// Mitsubishi GX Works2 project: plc_fact_fuc_1008   PLC: Q02/Q02H

// global labels: Global1
VAR_GLOBAL
  vision AT D100 : INT;
  scan AT D102 : INT;
END_VAR

PROGRAM MAIN
VAR
  CY_1 : pusher;
  CY_2 : pusher;
  CY_3 : pusher;
END_VAR
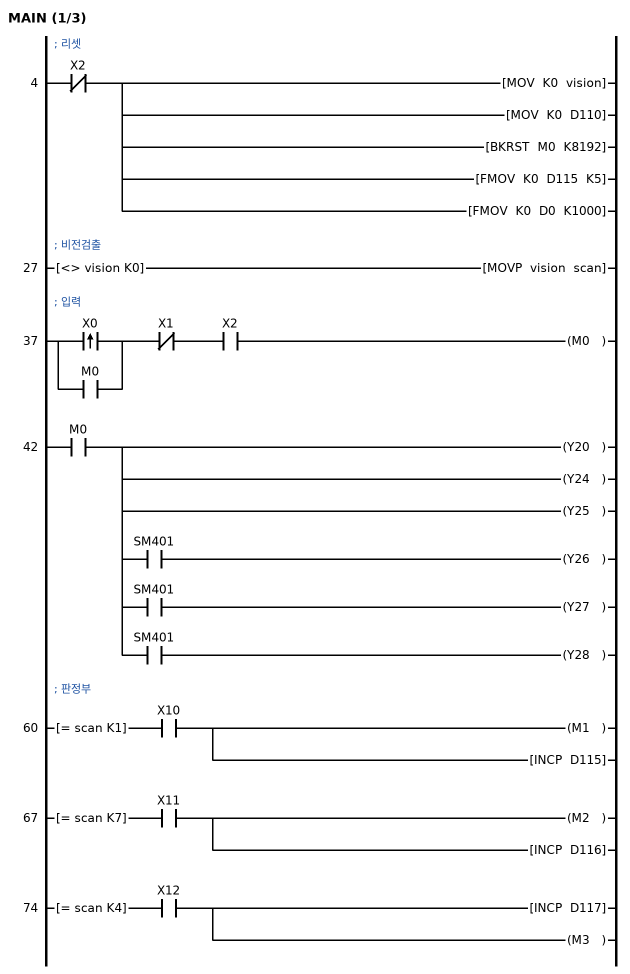
; 리셋
4     LDI     X2
      MOV     K0 vision
      MOV     K0 D110
      BKRST   M0 K8192
      FMOV    K0 D115 K5
      FMOV    K0 D0 K1000
; 비전검출
27    LD<>    vision K0
      MOVP    vision scan
; 입력
37    LDP     X0
      OR      M0
      ANI     X1
      AND     X2
      OUT     M0
42    LD      M0
      OUT     Y20
      OUT     Y24
      OUT     Y25
      MPS
      AND     SM401
      OUT     Y26
      MRD
      AND     SM401
      OUT     Y27
      MPP
      AND     SM401
      OUT     Y28
; 판정부
60    LD=     scan K1
      AND     X10
      OUT     M1
      INCP    D115
67    LD=     scan K7
      AND     X11
      OUT     M2
      INCP    D116
74    LD=     scan K4
      AND     X12
      INCP    D117
      OUT     M3
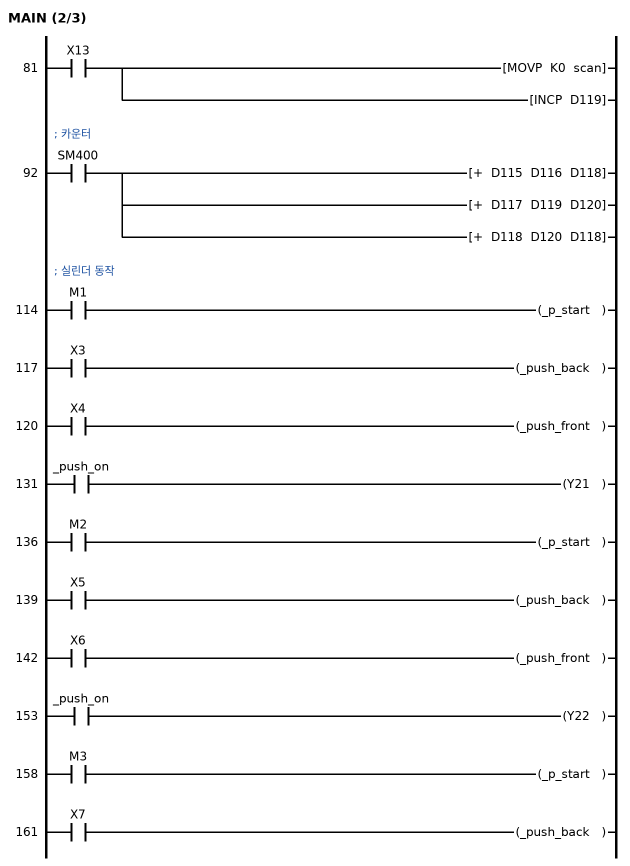
81    LD      X13
      MOVP    K0 scan
      INCP    D119
; 카운터
92    LD      SM400
      +       D115 D116 D118
      +       D117 D119 D120
      +       D118 D120 D118
; 실린더 동작
; FB BLK START pusher(CY_1)
114   LD      M1
      OUT     _p_start
117   LD      X3
      OUT     _push_back
120   LD      X4
      OUT     _push_front
; FB START
; FB_NAME pusher
; INSTANCE_NAME CY_1
; FB IN_B:p_start
; FB OUT_push_on:B
; FB IN_B:push_back
; FB IN_B:push_front
; FB END
131   LD      _push_on
      OUT     Y21
; FB BLK END
; FB BLK START pusher(CY_2)
136   LD      M2
      OUT     _p_start
139   LD      X5
      OUT     _push_back
142   LD      X6
      OUT     _push_front
; FB START
; FB_NAME pusher
; INSTANCE_NAME CY_2
; FB IN_B:p_start
; FB OUT_push_on:B
; FB IN_B:push_back
; FB IN_B:push_front
; FB END
153   LD      _push_on
      OUT     Y22
; FB BLK END
; FB BLK START pusher(CY_3)
158   LD      M3
      OUT     _p_start
161   LD      X7
      OUT     _push_back
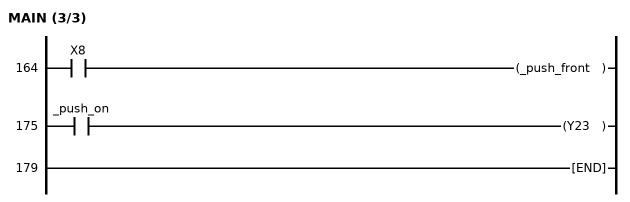
164   LD      X8
      OUT     _push_front
; FB START
; FB_NAME pusher
; INSTANCE_NAME CY_3
; FB IN_B:p_start
; FB OUT_push_on:B
; FB IN_B:push_back
; FB IN_B:push_front
; FB END
175   LD      _push_on
      OUT     Y23
; FB BLK END
179   END
END_PROGRAM

FUNCTION_BLOCK pusher
VAR_INPUT
  p_start : BOOL;
END_VAR
VAR
  pusher_timer : TIMER;
END_VAR
VAR_OUTPUT
  push_on : BOOL;
END_VAR
VAR
  MM1 : BOOL;
END_VAR
VAR_INPUT
  push_back : BOOL;
  push_front : BOOL;
END_VAR
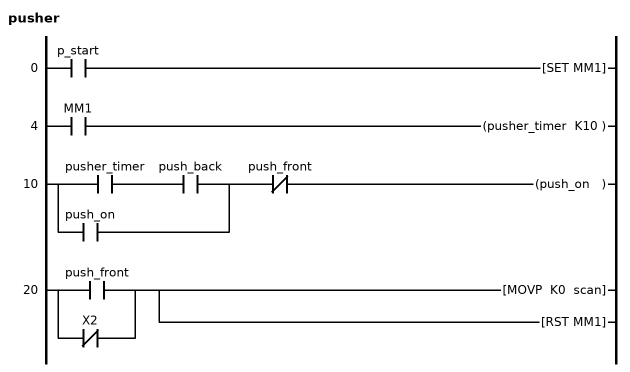
0     LD      p_start
      SET     MM1
4     LD      MM1
      OUT     pusher_timer K10
10    LD      pusher_timer
      AND     push_back
      OR      push_on
      ANI     push_front
      OUT     push_on
20    LD      push_front
      ORI     X2
      MOVP    K0 scan
      RST     MM1
END_FUNCTION_BLOCK
